(*

.. <legal notes>

legal notes
=================
| SPDX-FileCopyrightText: © 2026 Oleksandr Tiutyk <trofimich@gmail.com>
| SPDX-License-Identifier: LGPL-3.0-only
| For details check: LGPL-3.0-only_

.. _LGPL-3.0-only: https://www.gnu.org/licenses/lgpl-3.0.en.html

.. </legal notes>

*)

INTERFACE ICylinder EXTENDS Automation.ICompositeDevice

METHOD PUBLIC Extend
END_METHOD

{attribute 'monitoring' := 'call'}
{attribute 'OPC.UA.DA' := '1'}
{attribute 'OPC.UA.DA.Access' := '1'}
PROPERTY Extended : BOOL
GET
END_GET
END_PROPERTY

{attribute 'monitoring' := 'call'}
PROPERTY ExtendedInputContactType : CONTACT_TYPE
GET
END_GET
SET
END_SET
END_PROPERTY

{attribute 'monitoring' := 'call'}
{attribute 'OPC.UA.DA' := '1'}
{attribute 'OPC.UA.DA.Access' := '1'}
PROPERTY Extending : BOOL
GET
END_GET
END_PROPERTY

{attribute 'monitoring' := 'call'}
{attribute 'OPC.UA.DA' := '1'}
PROPERTY ExtendOutputContactType : CONTACT_TYPE
GET
END_GET
SET
END_SET
END_PROPERTY

{attribute 'monitoring' := 'call'}
{attribute 'OPC.UA.DA' := '1'}
PROPERTY HoldExtendOutput : BOOL
GET
END_GET
SET
END_SET
END_PROPERTY

{attribute 'monitoring' := 'call'}
{attribute 'OPC.UA.DA' := '1'}
PROPERTY HoldRetractOutput : BOOL
GET
END_GET
SET
END_SET
END_PROPERTY

{attribute 'TcRpcEnable':='1'}
METHOD PUBLIC Retract
END_METHOD

{attribute 'monitoring' := 'call'}
{attribute 'OPC.UA.DA' := '1'}
{attribute 'OPC.UA.DA.Access' := '1'}
PROPERTY Retracted : BOOL
GET
END_GET
END_PROPERTY

{attribute 'monitoring' := 'call'}
{attribute 'OPC.UA.DA' := '1'}
PROPERTY RetractedInputContactType : CONTACT_TYPE
GET
END_GET
SET
END_SET
END_PROPERTY

{attribute 'monitoring' := 'call'}
{attribute 'OPC.UA.DA' := '1'}
{attribute 'OPC.UA.DA.Access' := '1'}
PROPERTY Retracting : BOOL
GET
END_GET
END_PROPERTY

{attribute 'monitoring' := 'call'}
{attribute 'OPC.UA.DA' := '1'}
PROPERTY RetractOutputContactType : CONTACT_TYPE
GET
END_GET
SET
END_SET
END_PROPERTY

{attribute 'TcRpcEnable':='1'}
METHOD PUBLIC Stop
END_METHOD

END_INTERFACE

(* stored: Version 1.1.0.1
   Itf ICylinder: Id {31545994-a2c7-424b-9206-f5d8b74e123d}
   Folder Commands: Id {24e3800e-87bd-46d9-864c-0bcd101c50fa}
   Folder Settings: Id {65a64de5-9158-40ca-bc7c-ec332116d14f}
   Folder Statuses: Id {2472f38d-c571-4747-869b-1ac3231af82c}
   Method Extend: Id {cfd378ad-bc2f-4660-8ebd-9dfaa9315f24}
   Property Extended: Id {ac5e751e-f662-4074-babd-34dd772013fb}
   Get Get: Id {9f5f77e3-f332-4090-a8d1-aa5c025f4afc}
   Property ExtendedInputContactType: Id {20090080-3249-4987-839d-8560b88a4470}
   Get Get: Id {1efea601-ca15-43a0-8646-44c753626254}
   Set Set: Id {927c1d7b-2041-4880-86c0-0124bf2aba19}
   Property Extending: Id {6e79d079-3da3-4182-9977-b6630cf3bd44}
   Get Get: Id {9bc673c9-700b-4b6c-95e5-df1be254172a}
   Property ExtendOutputContactType: Id {b304a45b-759d-43c4-a81f-2d11516fd150}
   Get Get: Id {bee8c02d-eb22-44d0-b632-cd3e6aa5412a}
   Set Set: Id {8c23d9b5-1c22-476a-8a78-c8337b9daca3}
   Property HoldExtendOutput: Id {a269613f-ab98-467b-acd6-49259591d86e}
   Get Get: Id {b716d4a1-68a7-45cf-a1ea-e66cab3e1632}
   Set Set: Id {1f2ddffc-e1b5-45f9-ba1c-76212e1ed42b}
   Property HoldRetractOutput: Id {3918ac60-f216-4fa5-ad4a-db0a7d253672}
   Get Get: Id {f843aa1f-4f9f-4115-824a-75d5a6d3c970}
   Set Set: Id {0dae8609-4ef2-45b1-8594-8753ede34b47}
   Method Retract: Id {72cea106-046d-4616-b086-83f533a5f98b}
   Property Retracted: Id {49abf512-5008-4f85-a167-69120376ec6d}
   Get Get: Id {b9b01a8b-8870-4dc3-8b51-255374911e90}
   Property RetractedInputContactType: Id {804144d0-367d-441e-9dcc-79c7335b16a1}
   Get Get: Id {3f8da0e6-8f8f-4da6-b76b-d5b20ff8d5ef}
   Set Set: Id {983a44ea-c451-43b4-8cbf-17dbc504550b}
   Property Retracting: Id {83db92eb-f293-46bf-a0ad-a0d6ba56eca6}
   Get Get: Id {d26e06ef-22c1-4233-af15-a20cf398cc2a}
   Property RetractOutputContactType: Id {bcdedb62-dbcb-4b0c-9d99-9f76ecf54aa0}
   Get Get: Id {58c58d94-b59b-4318-8c15-3d5fa0d776f5}
   Set Set: Id {12b5c467-be00-4147-a311-e6003e679b3e}
   Method Stop: Id {ea3d2231-9b24-452d-b2c3-f49d196a7032} *)
